FUNCTION_BLOCK DACylCtlST (* Basic Function Block Type *)
  (* Standard: 61499-2 *)
  (* Version 0.0, 5/26/2016, Andrei, nxtControl GmbH, Template *)
  PACKAGE Main;
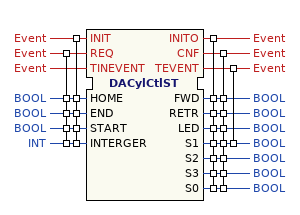
  EVENT_INPUT
    INIT WITH HOME, END, START, INTERGER; (* Initialization Request *)
    REQ WITH HOME, END, START, INTERGER; (* Normal Execution Request *)
    TINEVENT;
  END_EVENT
  EVENT_OUTPUT
    INITO WITH FWD, RETR, LED, S1, S2, S3, S0; (* Initialization Confirm *)
    CNF WITH FWD, RETR, LED, S1, S2, S3, S0; (* Execution Confirmation *)
    TEVENT WITH S1;
  END_EVENT
  VAR_INPUT
    HOME : BOOL; (* Input event qualifier *)
    END : BOOL;
    START : BOOL;
    INTERGER : INT;
  END_VAR
  VAR_OUTPUT
    FWD : BOOL;
    RETR : BOOL;
    LED : BOOL;
    S1 : BOOL;
    S2 : BOOL;
    S3 : BOOL;
    S0 : BOOL;
  END_VAR
  VAR
    State : INT;
    S1x : BOOL;
    S2x : BOOL;
    S3x : BOOL;
    S0x : BOOL;
    T1 : INT;
    T2 : INT;
  END_VAR
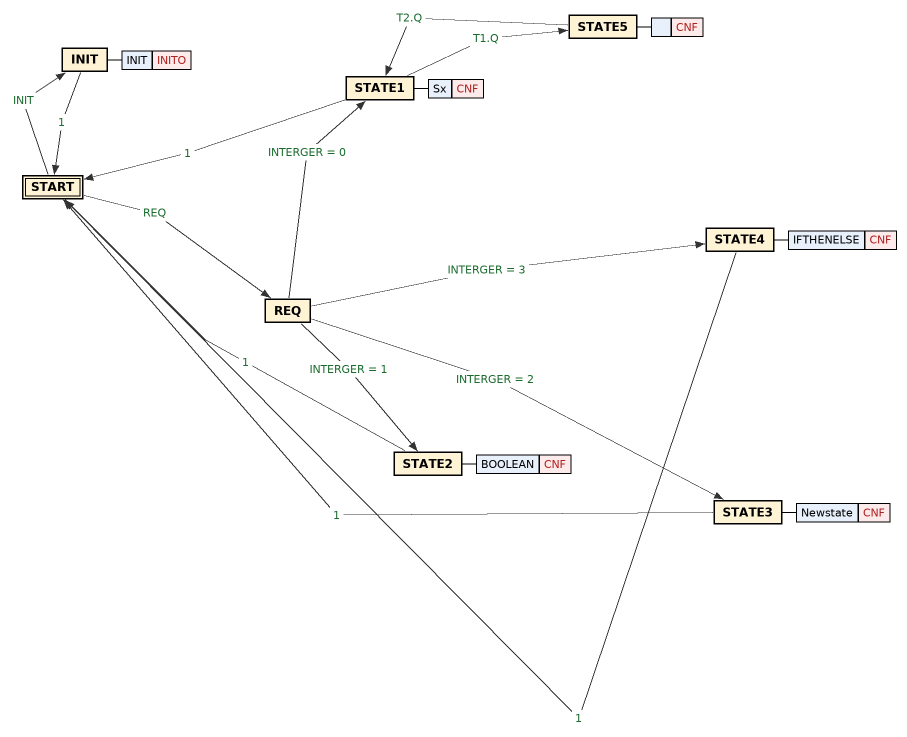
  EC_STATES
    START; (* Initial State *)
    REQ;
    INIT : INIT -> INITO;
    STATE1 : Sx -> CNF;
    STATE2 : BOOLEAN -> CNF;
    STATE3 : Newstate -> CNF;
    STATE4 : IFTHENELSE -> CNF;
    STATE5 : -> CNF;
  END_STATES
  EC_TRANSITIONS
    START TO INIT := INIT;
    START TO REQ := REQ;
    INIT TO START := 1;
    REQ TO STATE1 := INTERGER = 0;
    REQ TO STATE2 := INTERGER = 1;
    STATE2 TO START := 1;
    STATE1 TO START := 1;
    REQ TO STATE3 := INTERGER = 2;
    STATE3 TO START := 1;
    REQ TO STATE4 := INTERGER = 3;
    STATE4 TO START := 1;
    STATE5 TO STATE1 := T2.Q;
    STATE1 TO STATE5 := T1.Q;
  END_TRANSITIONS
  ALGORITHM INIT IN ST: (* Initialization algorithm *)
FWD :=FALSE;
RETR:=FALSE;
LED :=FALSE;
IF INTERGER >1 THEN
	S0 := TRUE;
	S1 := FALSE;
	S2 := FALSE;
	S3 := FALSE;
ELSE;
	S1 := TRUE;
	S2 := FALSE;
	S3 := FALSE;
END_IF;
  END_ALGORITHM
  ALGORITHM Sx IN ST:
S1x := 1;
S2x := 0;
S3x := 0;
S2x := S2 AND NOT END OR S1 AND START;
S3x := S3 AND NOT HOME OR S2 AND END;
S1x := S1 AND NOT START OR S3 AND HOME;
// Outputs
LED := S1x;
FWD := S2x;
RETR := S3x;
S1 := S1x;
S2 := S2x;
S3 := S3x;
  END_ALGORITHM
  ALGORITHM BOOLEAN IN ST:
S2:=S2 AND NOT END OR S1 AND START;
S3:=S3 AND NOT HOME OR S2 AND END;
S1:=S1 AND NOT START OR S3 AND HOME;

// Outputs
LED := S1;
FWD := S2;
RETR := S3;
  END_ALGORITHM
  ALGORITHM IFTHENELSE IN ST:
;

IF State=0 THEN
	LED:=FALSE;
	IF HOME THEN
		State:=1;
	END_IF;
ELSIF State = 1 THEN
	RETR:= FALSE;
	LED:=TRUE;
	IF START THEN
		State:=2;
	END_IF;
ELSIF State=2 THEN
	FWD:=TRUE;
	IF END THEN
		State:=3;
	END_IF;
ELSIF State=3 THEN
	RETR := TRUE;
	FWD := FALSE;
	RETR:=TRUE;
	IF HOME THEN
		State:=1;
	END_IF;
END_IF;
  END_ALGORITHM
  ALGORITHM Newstate IN ST:
;

	S2x := S2 AND NOT END OR S1 AND START;
	S3x := S3 AND NOT HOME OR S2 AND END;
	S1x := S1 AND NOT START OR S3 AND HOME OR S0 AND HOME;
	S0x := S0 AND NOT HOME;

	LED := S1x;
	FWD := S2x;
	RETR := S3x;
	S0 := S0x;
	S1 := S1x;
	S2 := S2x;
	S3 := S3x;
  END_ALGORITHM
  ALGORITHM Blinking IN ST:
;
  END_ALGORITHM
END_FUNCTION_BLOCK
